(* PLC project ARR NG V1.0, SoMachine Motion Logic Builder V1.56.49.0, author SESA100920 *)
(* stored: creationDateTime 2020-05-27T13:43:00.917405, version 0.0.0.0, modificationDateTime 2020-05-26T17:23:23.8723846 *)

PROGRAM ObjectSpawner
  VAR
    sIp : STRING(15) := '172.27.128.188';
    uiPort : UINT := 5006;
    fbUdpPeer : TCPUDP.FB_UDPPeer;
    stStringToSend : STRING;
    stX : STRING;
    stY : STRING;
    stID : STRING;
    stProduct : STRING;
    udiSize : UDINT;
    iCounter : INT := 1;
    iBeginCounter : INT := 1;
    bFirstProductActive : BOOL;
    iVal : INT;
  END_VAR

            IF iCounter >= g_c_uiNrOfLocations THEN
	iCounter := 1;
END_IF

CASE iVal OF
	0: IF fbUdpPeer.Open() THEN
		iVal := 1;
		END_IF
	1: 
		IF g_astPickLocations[1].astLocations[iCounter].lrActMCPosX <> 0 AND g_astPickLocations[1].astLocations[iCounter].lrActMCPosX > 0 THEN
			stID := CONCAT('ID', INT_TO_STRING(iCounter));
			stX := CONCAT('X', INT_TO_STRING(LREAL_TO_INT(g_astPickLocations[1].astLocations[iCounter].lrActMCPosX)));
			stY := CONCAT('Y', INT_TO_STRING(LREAL_TO_INT(g_astPickLocations[1].astLocations[iCounter].lrActMCPosY)));
			stStringToSend := CONCAT(stID, CONCAT(stX, stY));
			udiSize := SIZEOF(stStringToSend);
			fbUdpPeer.SendTo(sIp, uiPort, ADR(stStringToSend), udiSize);
			iCounter := iCounter + 1;
		ELSIF g_astPickLocations[1].astLocations[iBeginCounter].lrActMCPosX = 0 THEN
			iVal := 2;
			iCounter := iBeginCounter;
		ELSE
			iCounter := iBeginCounter;
		END_IF
	2: 
		IF g_astPickLocations[1].astLocations[iCounter].lrActMCPosX = 0 AND bFirstProductActive = TRUE THEN
			iCounter := iCounter + 1;
		ELSE
			iBeginCounter := iCounter;
			iVal := 1;
		END_IF
		
END_CASE
		
		IF g_astPickLocations[1].astLocations[1].lrActMCPosX <> 0 THEN
			bFirstProductActive := TRUE;
		END_IF
          
END_PROGRAM
